(* IEC 61131-3 sources: Trae_CLoudTest/_archive/2026-04-25_全局规范修订V4.1.0/旧版程序文件 (part 2) *)

(* ---- FB_打胶机送料机构_V4.0.0.st ---- *)
//==============================================================================
// 边框缓存机 PLC程序 - 打胶机送料机构纯逻辑功能块
// 版本: V4.0.0
// 项目: DJ-2026-005 边框缓存机
// 编制日期: 2026-04-23
// 遵循规范: IEC 61131-3, 810_PLC编程规范_DEV-V1.0.0
// 说明: 纯逻辑功能块 - 打胶机送料机构独立控制(不包含任何X/Y/M/D地址引用)
//       所有输入来自主控(已映射的逻辑变量), 所有输出给主控(由主控映射到Y地址)
//
// 核心工艺:
//   接收取放料机构的放料完成信号后, X2轴移动到打胶机取料位置
//   等待打胶机允许送料 -> 发送允许抓料信号 -> 等待打胶机取料完成
//   返回待机位置, 循环执行
//
// 架构特点:
//   - 纯逻辑块: 不包含任何X/Y/M/D地址引用
//   - 数据解耦: 通过逻辑变量接口与主控交互
//   - 6步状态机: 完整的自动送料循环控制
//   - 故障安全: 内置超时保护、伺服故障检测、安全区冲突检测
//   - 安全区管理: 与取放料机构的区域互锁, 防止机械碰撞
//   - 完全自包含, 无外部物理地址依赖
//==============================================================================

//==============================================================================
// 功能块: FB_1004_GlueMachineFeeder_BufferFraming - 打胶机送料机构纯逻辑控制
// 功能:
//   1. 自动模式状态机(6步完整送料循环)
//   2. 手动模式控制(X2轴点动前/后)
//   3. 初始化流程(伺服使能、状态清零)
//   4. 块内报警检测与处理(5种报警类型, 201~299段)
//   5. 安全区逻辑(与取放料机构的区域互锁)
//   6. 完全自包含, 无外部物理地址依赖
//==============================================================================
FUNCTION_BLOCK FB_1004_GlueMachineFeeder_BufferFraming

VAR_INPUT
    (*==========================================================================
      一、系统控制信号 (来自主控/HMI M区)
      ==========================================================================*)
    i_b使能               : BOOL;    // 总使能信号(主控系统就绪后置位)

    (*-------------------------------------------------------------------------
      模式选择 (互斥信号,来自HMI M区)
      -------------------------------------------------------------------------*)
    i_b自动模式           : BOOL;    // 自动运行模式选择
    i_b手动模式           : BOOL;    // 手动调试模式选择

    (*-------------------------------------------------------------------------
      操作按钮 (来自HMI,边沿触发或电平有效)
      -------------------------------------------------------------------------*)
    i_b启动               : BOOL;    // 自动循环启动按钮(上升沿触发)
    i_b停止               : BOOL;    // 自动循环停止按钮(电平有效)
    i_b复位               : BOOL;    // 故障复位/初始化按钮(电平有效)

    (*==========================================================================
      二、手动操作信号 (2个BOOL,来自HMI)
      注: 本功能块仅控制X2轴(打胶机送料方向的水平轴)
      ==========================================================================*)
    (*--- X2轴伺服点动控制 (2个) ---*)
    i_bX2轴点动前         : BOOL;    // 手动-X2轴向前点动(去打胶机取料位置方向)
    i_bX2轴点动后         : BOOL;    // 手动-X2轴向后点动(返回待机位置方向)

    (*==========================================================================
      三、工艺参数 (来自HMI设定或配方, REAL类型)
      ==========================================================================*)
    i_r送料速度           : REAL;    // X2轴送料运动速度(mm/s或%)
    i_r待机位置           : REAL;    // X2轴待机位置坐标(mm, 安全等待位置)
    i_r取料位置           : REAL;    // X2轴取料位置坐标(mm, 打胶机取料口位置)

    (*==========================================================================
      四、传感器输入 (4个BOOL,全部来自主控IO映射)
      注: 本功能块不直接读取X地址, 所有传感器由主控映射后传入
      仅涉及X2轴相关传感器
      ==========================================================================*)
    (*--- X2轴伺服状态信号 ---*)
    i_bX2轴_原点           : BOOL;    // X2轴伺服原点信号(Home/ORG)
    i_bX2轴_正向限位       : BOOL;    // X2轴正向限位(去打胶机侧限位)
    i_bX2轴_反向限位       : BOOL;    // X2轴反向限位(待机位侧限位)
    i_bX2轴_伺服故障       : BOOL;    // X2轴伺服驱动器故障(ALM输出)

    (*==========================================================================
      五、打胶机交互信号 (2个BOOL,已由主控做IO映射)
      注: 这些是来自外部打胶机的硬接线信号, 由主控完成IO映射
      ==========================================================================*)
    i_b打胶机允许送料     : BOOL;    // 打胶机允许送料信号(对应物理地址X76)
                                    // TRUE=打胶机准备好可以接收边框
    i_b打胶机取料完成     : BOOL;    // 打胶机取料完成信号(对应物理地址X102)
                                    // TRUE=打胶机已完成边框抓取

    (*==========================================================================
      六、上游信号 (1个BOOL,来自取放料机构)
      ==========================================================================*)
    i_b取放料_放料完成    : BOOL;    // 取放料机构放料完成信号
                                    // TRUE=取放料机构已完成放料并移出安全区
END_VAR

VAR_OUTPUT
    (*==========================================================================
      一、执行器请求输出 (给主控, 由主控映射到Y地址)
      ==========================================================================*)

    (*--- 给打胶机的输出信号 ---*)
    o_b允许抓料            : BOOL;    // 允许抓料信号 -> 主控映射到Y44
                                    // 通知打胶机可以抓取边框(本站已到位且准备好)

    (*--- X2轴运动请求输出 (给主控驱动脉冲输出) ---*)
    o_bX2轴请求前移       : BOOL;    // X2轴向前移动请求(去打胶机取料位置)
    o_bX2轴请求后移       : BOOL;    // X2轴向后移动请求(返回待机位置)

    (*--- 安全区管理信号 ---*)
    o_b安全区信号          : BOOL;    // 安全区信号 -> 主控映射到Y47
                                    // TRUE=取放料机构在安全区外(打胶机可进入)
                                    // FALSE=取放料机构在工作区(禁止打胶机进入)

    (*==========================================================================
      二、状态/HMI显示输出
      ==========================================================================*)
    o_b运行中             : BOOL;    // 本站正在自动运行
    o_b故障               : BOOL;    // 本站有故障(任一报警激活)
    o_i当前状态           : INT;     // 当前状态机步序(0~5, 99=故障)
    o_rX2轴当前位置       : REAL;    // X2轴当前位置反馈(mm, 来自主控映射)

    (*==========================================================================
      三、报警输出 (给公共报警管理器)
      ==========================================================================*)
    o_i本站报警代码       : INT;     // 本站当前有效报警代码(0=无报警, 201~299=报警类型)
END_VAR

(*==============================================================================
 内部变量定义
 ==============================================================================*)
VAR
    (*--------------------------------------------------------------------------
      一、状态机核心变量
      --------------------------------------------------------------------------*)
    s_i步序               : INT;     // 当前状态机步序(0~5)
    s_b运行中             : BOOL;    // 自动运行中标志
    s_b故障               : BOOL;    // 故障标志
    s_b启动触发           : BOOL;    // 启动信号锁存(防重复触发)

    (*--- X2轴运动请求标志 (给主控处理脉冲输出) ---*)
    s_bX2轴请求前移       : BOOL;    // X2轴向前移动请求(去取料位置)
    s_bX2轴请求后移       : BOOL;    // X2轴向后移动请求(返回待机位置)
    s_bX2轴在待机位       : BOOL;    // X2轴是否在待机位置标志(由主控反馈)
    s_bX2轴在取料位       : BOOL;    // X2轴是否在取料位置标志(由主控反馈)

    (*--- 安全区管理变量 ---*)
    s_b取放料曾工作      : BOOL;    // 取放料机构曾经工作过标志(用于安全区判断)
    s_b上次放料完成      : BOOL;    // 上次扫描周期的放料完成状态(用于上升沿检测)

    (*--- 打胶机通讯超时检测 ---*)
    s_t通讯超时定时器     : TON;     // 打胶机响应超时检测定时器
    s_b等待打胶机响应     : BOOL;    // 正在等待打胶机响应标志

    (*--------------------------------------------------------------------------
      二、定时器 (覆盖所有时序需求)
      --------------------------------------------------------------------------*)
    s_t动作定时器         : TON;     // 通用动作等待定时器(X2轴移动等)
    s_t初始化定时器       : TON;     // 初始化总超时定时器
    s_t抓料保持定时器     : TON;     // 允许抓料信号保持定时器

    (*--------------------------------------------------------------------------
      三、系统级内部变量
      --------------------------------------------------------------------------*)
    s_b初始化完成         : BOOL;    // 上电初始化完成标志
    s_b初始化中           : BOOL;    // 正在执行初始化

    (*--- 报警相关 ---*)
    s_i活跃报警           : INT;     // 当前最高优先级报警代码

    (*--- 手动操作互锁 ---*)
    s_b手动允许           : BOOL;    // 允许手动操作标志
END_VAR

(*==============================================================================
 常量定义 (状态机步序 + 报警码 + 定时参数)
 ==============================================================================*)
VAR CONSTANT
    (*--------------------------------------------------------------------------
      状态机步序常量 (6步: 0空闲 + 5工作步)
      核心工艺: 接收放料完成 -> 移动到取料位 -> 等待允许 -> 抓料 -> 返回待机
      --------------------------------------------------------------------------*)
    STP_空闲              : INT := 0;   // 空闲/待机位置
    STP_等待放料完成      : INT := 1;   // 等待取放料机构放料完成
    STP_移动到取料位置    : INT := 2;   // X2轴移动到打胶机取料位置
    STP_等待允许送料      : INT := 3;   // 等待打胶机允许送料信号
    STP_发送允许抓料      : INT := 4;   // 发送允许抓料+等待打胶机取料完成
    STP_返回待机位置      : INT := 5;   // X2轴返回待机位置

    (*--------------------------------------------------------------------------
      报警码常量 (201~299段, 0=无报警)
      与取放料机构(101~199段)、其他设备错开, 便于公共报警管理器区分来源
      --------------------------------------------------------------------------*)
    ALM_通讯超时          : INT := 201;  // 通讯超时(打胶机无响应)
    ALM_安全区冲突        : INT := 202;  // 安全区冲突(取放料未离开)
    ALM_X2轴伺服故障      : INT := 203;  // X2轴伺服驱动器故障
    ALM_X2轴移动超时      : INT := 204;  // X2轴移动超时(未到达目标位置)
    ALM_取料位置到达超时  : INT := 205;  // 取料位置到达超时(步骤2专用)

    (*--------------------------------------------------------------------------
      默认定时参数 (单位: ms 或 s, 可通过输入参数覆盖)
      --------------------------------------------------------------------------*)
    T_DEF_移动超时时间    : INT := 5000;    // X2轴移动超时保护(5s)
    T_DEF_通讯超时时间    : INT := 10000;   // 打胶机响应超时(10s)
    T_DEF_抓料保持时间    : INT := 500;     // 允许抓料信号保持时间(500ms)
    T_DEF_初始化超时      : INT := 10000;   // 初始化总超时(10s)
END_VAR

(*==============================================================================
 主程序开始
 ==============================================================================*)

//==============================================================================
// 第一部分: 使能与初始化处理
//==============================================================================

(*--- 使能失效时的安全处理: 全部输出归零, 状态复位 ---*)
IF NOT i_b使能 THEN
    (
    (* 清零所有执行器输出 *)
    o_b允许抓料            := FALSE;
    o_b安全区信号          := FALSE;
    o_bX2轴请求前移       := FALSE;
    o_bX2轴请求后移       := FALSE;

    (* 清零所有状态 *)
    s_i步序               := STP_空闲
    s_b运行中             := FALSE;
    s_b故障               := FALSE;
    s_b启动触发           := FALSE;

    (* 清零运动请求 *)
    s_bX2轴请求前移       := FALSE;
    s_bX2轴请求后移       := FALSE;
    s_bX2轴在待机位       := FALSE;
    s_bX2轴在取料位       := FALSE;

    (* 清零安全区变量 *)
    s_b取放料曾工作      := FALSE;
    s_b上次放料完成      := FALSE;
    s_b等待打胶机响应     := FALSE;

    (* 清零报警 *)
    s_i活跃报警           := 0;
    o_i本站报警代码       := 0;
    o_b故障               := FALSE;
    s_b初始化完成         := FALSE;
    s_b初始化中           := FALSE;

    (* 清零状态输出 *)
    o_b运行中             := FALSE;
    o_i当前状态           := STP_空闲;

    (* 停止所有定时器 *)
    s_t动作定时器(IN := FALSE);
    s_t通讯超时定时器(IN := FALSE);
    s_t初始化定时器(IN := FALSE);
    s_t抓料保持定时器(IN := FALSE);

    RETURN;  (* 退出功能块, 不执行后续逻辑 *)
END_IF;

//==============================================================================
// 第二部分: 初始化流程 (上电或复位后首次使能时执行)
//==============================================================================

IF NOT s_b初始化完成 THEN
    s_b初始化中 := TRUE;

    (* 初始化定时器: 防止初始化卡死 *)
    s_t初始化定时器(IN := TRUE, PT := T_DEF_初始化超时);

    (* 初始化动作:
       1. 所有输出回到安全状态(禁止抓料, 安全区FALSE)
       2. 伺服使能准备(实际使能由主控统一协调)
       3. 状态清零
    *)

    (* 安全输出状态: 禁止抓料, 安全区默认FALSE(保守策略) *)
    o_b允许抓料            := FALSE;
    o_b安全区信号          := FALSE;
    o_bX2轴请求前移       := FALSE;
    o_bX2轴请求后移       := FALSE;

    (* 步序归零 *)
    s_i步序               := STP_空闲;
    s_b故障               := FALSE;
    s_i活跃报警           := 0;

    (* 检查初始化条件:
       X2轴伺服无故障 AND (已在原点 OR 超时强制完成)
       允许在有非关键报警情况下继续, 报警单独处理
    *)
    IF (NOT i_bX2轴_伺服故障) OR s_t初始化定时器.Q THEN
        (* 初始化完成 或 超时强制完成(伺服故障会单独报203号报警) *)
        s_b初始化完成 := TRUE;
        s_b初始化中 := FALSE;
        s_t初始化定时器(IN := FALSE);

        (* 初始化完成后关闭输出(进入空闲态的安全状态) *)
        o_b允许抓料        := FALSE;
        o_b安全区信号      := FALSE;
        o_bX2轴请求前移   := FALSE;
        o_bX2轴请求后移   := FALSE;
    END_IF;

    (* 初始化期间不执行自动/手动逻辑 *)
    o_b运行中 := FALSE;
    o_i当前状态 := STP_空闲;
    RETURN;
END_IF;

//==============================================================================
// 第三部分: 安全区逻辑处理 (所有模式共用, 最高优先级之一)
//==============================================================================

(*--- 安全区核心逻辑 ---
   目的: 防止取放料机构和打胶机同时在工作区域造成碰撞
   原则: 取放料机构优先(它是主动方, 先放料后打胶机才能进来)

   判断依据:
   - i_b取放料_放料完成 = TRUE 表示取放料机构已完成放料并移出工作区
   - 当取放料机构正在工作时(放料完成=FALSE), 安全区应为FALSE
   - 只有当放料完成且确认离开后, 安全区才为TRUE
*)

(*--- 检测取放料机构工作状态的上升沿 ---*)
(* 当放料完成从FALSE变为TRUE时, 说明取放料机构刚完成工作并离开 *)
IF i_b取放料_放料完成 AND NOT s_b上次放料完成 THEN
    (* 放料完成的上升沿: 标记取放料机构曾工作过, 现在已离开 *)
    s_b取放料曾工作 := TRUE;
ELSIF NOT i_b取放料_放料完成 THEN
    (* 放料完成=FALSE: 取放料机构可能正在工作中或尚未开始 *)
    (* 如果之前有过放料完成又变为FALSE, 说明新的一轮开始了 *)
END_IF;

(*--- 更新上次状态(用于下次扫描周期的上升沿检测) ---*)
s_b上次放料完成 := i_b取放料_放料完成;

(*--- 安全区信号输出逻辑 ---*)
IF i_b取放料_放料完成 THEN
    (* 放料完成=TRUE: 取放料机构已离开工作区, 安全区开放 *)
    o_b安全区信号 := TRUE;
ELSE
    (* 放料完成=FALSE: 取放料机构可能还在工作区, 安全区关闭 *)
    o_b安全区信号 := FALSE;
END_IF;

//==============================================================================
// 第四部分: X2轴伺服故障检测 (所有模式共用, 最高优先级)
//==============================================================================

(*--- X2轴伺服故障检测 ---*)
IF i_bX2轴_伺服故障 THEN
    IF s_i活跃报警 <> ALM_X2轴伺服故障 THEN
        (* 新故障: 记录报警 *)
        s_i活跃报警 := ALM_X2轴伺服故障;
        s_b故障 := TRUE;
    END_IF;
    (* 伺服故障时立即停止X2轴运动请求 *)
    s_bX2轴请求前移   := FALSE;
    o_bX2轴请求前移   := FALSE;
    s_bX2轴请求后移   := FALSE;
    o_bX2轴请求后移   := FALSE;
ELSIF s_i活跃报警 = ALM_X2轴伺服故障 THEN
    (* 故障消失且当前只有此报警 -> 清除 *)
    s_i活跃报警 := 0;
    s_b故障 := FALSE;
END_IF;

//==============================================================================
// 第五部分: 模式分发 (自动/手动)
//==============================================================================

IF i_b自动模式 THEN
    (*==========================================================================
      自动模式: 执行6步送料状态机
      =========================================================================*)
    CALL_自动模式状态机();

ELSIF i_b手动模式 THEN
    (*==========================================================================
      手动模式: 执行手动点动控制(X2轴前后点动)
      =========================================================================*)
    CALL_手动模式控制();

ELSE
    (* 无效模式: 停止所有输出, 进入安全状态 *)
    o_b允许抓料            := FALSE;
    o_bX2轴请求前移       := FALSE;
    o_bX2轴请求后移       := FALSE;

    (* 如果不在故障态, 归零步序 *)
    IF NOT s_b故障 THEN
        s_i步序 := STP_空闲;
        s_b运行中 := FALSE;
    END_IF;
END_IF;

//==============================================================================
// 第六部分: 停止与复位处理
//==============================================================================

(*--- 全局停止: 停止自动循环, 保持当前位置 ---*)
IF i_b停止 THEN
    IF s_b运行中 AND NOT s_b故障 THEN
        (* 停止并复位到空闲 *)
        s_i步序 := STP_空闲;
        s_b运行中 := FALSE;
        s_b启动触发 := FALSE;

        (* 停止所有输出 *)
        o_b允许抓料            := FALSE;
        o_bX2轴请求前移       := FALSE;
        o_bX2轴请求后移       := FALSE;
        s_bX2轴请求前移       := FALSE;
        s_bX2轴请求后移       := FALSE;

        (* 停止定时器 *)
        s_t动作定时器(IN := FALSE);
        s_t通讯超时定时器(IN := FALSE);
        s_t抓料保持定时器(IN := FALSE);
        s_b等待打胶机响应     := FALSE;
    END_IF;
END_IF;

(*--- 全局复位: 清除所有报警和故障, 重新初始化 ---*)
IF i_b复位 THEN
    IF s_b故障 THEN
        (* 清除报警和故障标志 *)
        s_i活跃报警 := 0;
        s_b故障 := FALSE;
        o_i本站报警代码 := 0;

        (* 归零步序和计数器 *)
        s_i步序 := STP_空闲;
        s_b运行中 := FALSE;
        s_b启动触发 := FALSE;

        (* 安全输出状态: 全部归零 *)
        o_b允许抓料            := FALSE;
        o_bX2轴请求前移       := FALSE;
        o_bX2轴请求后移       := FALSE;
        s_bX2轴请求前移       := FALSE;
        s_bX2轴请求后移       := FALSE;
        s_bX2轴在待机位       := FALSE;
        s_bX2轴在取料位       := FALSE;

        (* 清零安全区变量 *)
        s_b取放料曾工作      := FALSE;
        s_b等待打胶机响应     := FALSE;

        (* 停止定时器 *)
        s_t动作定时器(IN := FALSE);
        s_t通讯超时定时器(IN := FALSE);
        s_t抓料保持定时器(IN := FALSE);

        (* 要求重新初始化 *)
        s_b初始化完成 := FALSE;
    END_IF;
END_IF;

//==============================================================================
// 第七部分: 状态输出汇总
//==============================================================================

(*--- 运行中标志 ---*)
o_b运行中 := s_b运行中;

(*--- 故障标志 ---*)
o_b故障 := s_b故障;

(*--- 当前状态码 ---*)
IF s_b故障 THEN
    o_i当前状态 := 99;  (* 故障状态显示99 *)
ELSE
    o_i当前状态 := s_i步序;
END_IF;

(*--- 本站报警代码 ---*)
o_i本站报警代码 := s_i活跃报警;

(*==============================================================================
 子程序: 自动模式状态机 (6步完整送料循环)
   核心工艺: 等待放料完成 -> X2轴移动到取料位 -> 等待允许 -> 抓料 -> 返回待机
   安全约束: 步骤1需要安全区信号为TRUE才能继续
  ==============================================================================*)
METHOD CALL_自动模式状态机 : VOID

    (*--- 故障时不执行状态机 ---*)
    IF s_b故障 THEN
        s_b运行中 := FALSE;
        (* 故障安全输出: 全部停止 *)
        o_b允许抓料            := FALSE;
        o_bX2轴请求前移       := FALSE;
        o_bX2轴请求后移       := FALSE;
        s_bX2轴请求前移       := FALSE;
        s_bX2轴请求后移       := FALSE;
        s_t动作定时器(IN := FALSE);
        s_t通讯超时定时器(IN := FALSE);
        s_t抓料保持定时器(IN := FALSE);
        s_b等待打胶机响应     := FALSE;
        RETURN;
    END_IF;

    (*--- 启动触发检测 (上升沿) ---*)
    IF i_b启动 AND NOT s_b启动触发 THEN
        s_b启动触发 := TRUE;
    END_IF;

    (*--- 单例状态机 (全局唯一, 因为只有一个打胶机送料机构) ---*)
    CASE s_i步序 OF

    (*======================================================================
     步骤0: 空闲/待机位置
     等待启动触发, 收到启动后进入等待放料完成
     ======================================================================*)
    STP_空闲:
        s_b运行中 := FALSE;
        (* 安全输出状态: 全部归零 *)
        o_b允许抓料            := FALSE;
        o_bX2轴请求前移       := FALSE;
        o_bX2轴请求后移       := FALSE;
        s_bX2轴请求前移       := FALSE;
        s_bX2轴请求后移       := FALSE;
        s_b等待打胶机响应     := FALSE;

        (* 启动条件: 收到启动触发 *)
        IF s_b启动触发 THEN
            s_i步序 := STP_等待放料完成;
            s_b运行中 := TRUE;
        END_IF;

    (*======================================================================
     步骤1: 等待取放料放料完成
     等待取放料机构的放料完成信号(即安全区开放)
     条件: i_b取放料_放料完成 = TRUE
     ======================================================================*)
    STP_等待放料完成:
        (* 保持安全输出状态 *)
        o_b允许抓料            := FALSE;
        o_bX2轴请求前移       := FALSE;
        o_bX2轴请求后移       := FALSE;
        s_bX2轴请求前移       := FALSE;
        s_bX2轴请求后移       := FALSE;

        (* 等待条件: 取放料机构放料完成(安全区开放) *)
        IF i_b取放料_放料完成 THEN
            (* 放料完成, 可以开始移动到取料位置 *)
            s_i步序 := STP_移动到取料位置;
            (* 启动移动超时定时器 *)
            s_t动作定时器(IN := TRUE, PT := T_DEF_移动超时时间);
            (* 请求X2轴向前移动(去打胶机取料位置) *)
            s_bX2轴请求前移   := TRUE;
            o_bX2轴请求前移   := TRUE;
            s_bX2轴请求后移   := FALSE;
            o_bX2轴请求后移   := FALSE;
            s_bX2轴在待机位   := FALSE;
        END_IF;

        (* 注意: 此步骤没有独立的超时报警, 因为等待上游信号是正常行为
           超时保护由公共层或操作员手动停止处理 *)

    (*======================================================================
     步骤2: 移动到打胶机取料位置 (X2轴水平移动)
     X2轴向前移动到打胶机取料口位置
     等待X2轴到达取料位置或超时
     注: X2轴的实际脉冲输出由主控根据请求标志处理
     ======================================================================*)
    STP_移动到取料位置:
        (* 保持X2轴前移请求 *)
        s_bX2轴请求前移   := TRUE;
        o_bX2轴请求前移   := TRUE;
        s_bX2轴请求后移   := FALSE;
        o_bX2轴请求后移   := FALSE;

        (* 到达取料位置的判断:
           由主控在X2轴到达目标位置后置位s_bX2轴在取料位
           或通过位置判断(i_rX2轴当前位置接近i_r取料位置)
        *)
        IF s_bX2轴在取料位 THEN
            (* 到达取料位置, 转入等待打胶机允许送料 *)
            s_t动作定时器(IN := FALSE);
            s_bX2轴请求前移   := FALSE;
            o_bX2轴请求前移   := FALSE;
            s_bX2轴在取料位   := TRUE;
            s_i步序 := STP_等待允许送料;
            (* 启动通讯超时定时器(等待打胶机响应) *)
            s_t通讯超时定时器(IN := TRUE, PT := T_DEF_通讯超时时间);
            s_b等待打胶机响应 := TRUE;
        ELSIF s_t动作定时器.Q THEN
            (* 超时: X2轴未在规定时间内到达取料位置 *)
            s_t动作定时器(IN := FALSE);
            s_i活跃报警 := ALM_X2轴移动超时;
            s_b故障 := TRUE;
            s_bX2轴请求前移   := FALSE;
            o_bX2轴请求前移   := FALSE;
            s_i步序 := STP_空闲;
            s_b运行中 := FALSE;
            s_b启动触发 := FALSE;
            s_b等待打胶机响应 := FALSE;
        END_IF;

    (*======================================================================
     步骤3: 等待打胶机允许送料
     等待打胶机发出允许送料信号(i_b打胶机允许送料=TRUE)
     同时监控通讯超时
     ======================================================================*)
    STP_等待允许送料:
        (* 保持当前状态, 等待打胶机响应 *)
        s_bX2轴请求前移   := FALSE;
        o_bX2轴请求前移   := FALSE;
        s_bX2轴请求后移   := FALSE;
        o_bX2轴请求后移   := FALSE;
        o_b允许抓料        := FALSE;

        (* 检查打胶机允许送料信号 *)
        IF i_b打胶机允许送料 THEN
            (* 打胶机允许送料, 转入发送允许抓料步骤 *)
            s_t通讯超时定时器(IN := FALSE);
            s_b等待打胶机响应 := FALSE;
            s_i步序 := STP_发送允许抓料;
            (* 启动抓料保持定时器和通讯超时定时器(等待取料完成) *)
            s_t抓料保持定时器(IN := TRUE, PT := T_DEF_抓料保持时间);
            s_t通讯超时定时器(IN := TRUE, PT := T_DEF_通讯超时时间);
            s_b等待打胶机响应 := TRUE;
            (* 发送允许抓料信号 *)
            o_b允许抓料 := TRUE;
        ELSIF s_t通讯超时定时器.Q THEN
            (* 超时: 打胶机长时间无响应 *)
            s_t通讯超时定时器(IN := FALSE);
            s_i活跃报警 := ALM_通讯超时;
            s_b故障 := TRUE;
            o_b允许抓料 := FALSE;
            s_b等待打胶机响应 := FALSE;
            s_i步序 := STP_空闲;
            s_b运行中 := FALSE;
            s_b启动触发 := FALSE;
        END_IF;

    (*======================================================================
     步骤4: 发送允许抓料 + 等待打胶机取料完成
     保持允许抓料信号, 等待打胶机完成取料动作
     ======================================================================*)
    STP_发送允许抓料:
        (* 保持允许抓料输出 *)
        o_b允许抓料 := TRUE;
        s_bX2轴请求前移 := FALSE;
        o_bX2轴请求前移 := FALSE;
        s_bX2轴请求后移 := FALSE;
        o_bX2轴请求后移 := FALSE;

        (* 检查打胶机取料完成信号 *)
        IF i_b打胶机取料完成 THEN
            (* 打胶机取料完成, 转入返回待机位置 *)
            s_t通讯超时定时器(IN := FALSE);
            s_t抓料保持定时器(IN := FALSE);
            s_b等待打胶机响应 := FALSE;
            (* 保持一段时间的允许抓料信号后关闭 *)
            (* 或者立即关闭, 根据实际工艺需求 *)
            o_b允许抓料 := FALSE;
            s_i步序 := STP_返回待机位置;
            (* 启动返回移动定时器 *)
            s_t动作定时器(IN := TRUE, PT := T_DEF_移动超时时间);
            (* 请求X2轴向后移动(返回待机位置) *)
            s_bX2轴请求前移   := FALSE;
            o_bX2轴请求前移   := FALSE;
            s_bX2轴请求后移   := TRUE;
            o_bX2轴请求后移   := TRUE;
            s_bX2轴在取料位   := FALSE;
        ELSIF s_t通讯超时定时器.Q THEN
            (* 超时: 打胶机取料超时 *)
            s_t通讯超时定时器(IN := FALSE);
            s_t抓料保持定时器(IN := FALSE);
            s_i活跃报警 := ALM_通讯超时;
            s_b故障 := TRUE;
            o_b允许抓料 := FALSE;
            s_b等待打胶机响应 := FALSE;
            s_bX2轴请求后移 := FALSE;
            o_bX2轴请求后移 := FALSE;
            s_i步序 := STP_空闲;
            s_b运行中 := FALSE;
            s_b启动触发 := FALSE;
        END_IF;

    (*======================================================================
     步骤5: 返回待机位置 (X2轴水平移动回待机位)
     X2轴向后移动回到待机位置(安全等待位置)
     等待X2轴到达待机位置或超时
     完成后回到步骤1, 继续下一轮循环
     ======================================================================*)
    STP_返回待机位置:
        (* 保持X2轴后移请求 *)
        s_bX2轴请求前移   := FALSE;
        o_bX2轴请求前移   := FALSE;
        s_bX2轴请求后移   := TRUE;
        o_bX2轴请求后移   := TRUE;

        (* 到达待机位置的判断:
           由主控在X2轴到达目标位置后置位s_bX2轴在待机位
           或通过位置判断(i_rX2轴当前位置接近i_r待机位置)
        *)
        IF s_bX2轴在待机位 THEN
            (* 到达待机位置, 完成一轮循环, 回到等待放料完成 *)
            s_t动作定时器(IN := FALSE);
            s_bX2轴请求后移   := FALSE;
            o_bX2轴请求后移   := FALSE;
            s_bX2轴在待机位   := TRUE;
            s_i步序 := STP_等待放料完成;  (* 回到步骤1, 继续循环 *)
            (* 不重置s_b启动触发, 保持连续循环 *)
        ELSIF s_t动作定时器.Q THEN
            (* 超时: X2轴未在规定时间内返回待机位置 *)
            s_t动作定时器(IN := FALSE);
            s_i活跃报警 := ALM_X2轴移动超时;
            s_b故障 := TRUE;
            s_bX2轴请求后移   := FALSE;
            o_bX2轴请求后移   := FALSE;
            s_i步序 := STP_空闲;
            s_b运行中 := FALSE;
            s_b启动触发 := FALSE;
        END_IF;

    ELSE
        (* 无效步序: 强制归零 *)
        s_i步序 := STP_空闲;
        s_b运行中 := FALSE;

    END_CASE;

(*==============================================================================
 子程序: 手动模式控制 (X2轴点动前/后, 带互锁和安全限制)
  ==============================================================================*)
METHOD CALL_手动模式控制 : VOID

    (*--- 故障时禁止手动操作 ---*)
    IF s_b故障 THEN
        s_b手动允许 := FALSE;
        o_b允许抓料            := FALSE;
        s_bX2轴请求前移       := FALSE;
        s_bX2轴请求后移       := FALSE;
        s_i步序 := STP_空闲;
        s_b运行中 := FALSE;
        RETURN;
    END_IF;

    s_b手动允许 := TRUE;
    s_b运行中 := FALSE;
    s_i步序 := STP_空闲;  (* 手动模式下步序显示为空闲 *)
    o_b允许抓料 := FALSE;   (* 手动模式下不允许自动抓料 *)

    (*======================================================================
     手动操作 - X2轴伺服点动控制 (前/后互锁)
     注意: 伺服的点动脉冲输出由主控根据请求标志处理
     本功能块只输出请求标志
     ======================================================================*)

    (*--- X2轴点动: 前/后互锁 ---*)
    IF i_bX2轴点动前 AND NOT i_bX2轴点动后 THEN
        (* X2轴向前点动(去打胶机取料位置方向) *)
        (* 检查是否已到正向限位 *)
        IF NOT i_bX2轴_正向限位 THEN
            s_bX2轴请求前移 := TRUE;
            o_bX2轴请求前移 := TRUE;
            s_bX2轴请求后移 := FALSE;
            o_bX2轴请求后移 := FALSE;
        END_IF;
    ELSIF i_bX2轴点动后 AND NOT i_bX2轴点动前 THEN
        (* X2轴向后点动(返回待机位置方向) *)
        (* 检查是否已到反向限位 *)
        IF NOT i_bX2轴_反向限位 THEN
            s_bX2轴请求后移 := TRUE;
            o_bX2轴请求后移 := TRUE;
            s_bX2轴请求前移 := FALSE;
            o_bX2轴请求前移 := FALSE;
        END_IF;
    ELSE
        (* 无X2轴点动操作 *)
        s_bX2轴请求前移 := FALSE;
        o_bX2轴请求前移 := FALSE;
        s_bX2轴请求后移 := FALSE;
        o_bX2轴请求后移 := FALSE;
    END_IF;

END_FUNCTION_BLOCK

//==============================================================================
// 程序结束
//==============================================================================

(* ---- 主控程序_V4.0.0.st ---- *)
//==============================================================================
// 边框缓存机 PLC程序 - 主控程序 (V4.0.0架构)
// 版本: V4.0.0
// 项目: DJ-2026-005 边框缓存机
// 编制日期: 2026-04-23
// 更新日期: 2026-04-24 (新增打胶机/组框机交互接口预留)
// 遵循规范: IEC 61131-3, 810_PLC编程规范_DEV-V1.0.0
//
// 说明:
//   主控程序是系统的核心协调组件,承担以下职责:
//   1. IO映射: X地址->逻辑变量(传感器输入), 逻辑变量->Y地址(执行器输出)
//   2. HMI数据交互: M/D区读取(操作指令/参数设定), M/D区回写(状态/报警)
//   3. 外部设备交互:
//      - 下游打胶机: 允许送料(X76), 取料完成(X102), 故障/急停联锁
//      - 上游组框机: 允许送料, 有料请求, 开门互锁, 安全联锁 (预留接口)
//   4. 工站实例化与连接: 实例化4个功能块并按工艺顺序调用
//   5. 报警汇总: 调用公共报警管理器,汇总三工站报警并写入D区
//
// 架构特点:
//   - 纯协调层: 不包含任何业务逻辑(状态机/自动手动判断在工站内部)
//   - 数据桥梁: 连接物理IO层(X/Y)与逻辑层(功能块接口变量)
//   - 设备协调: 处理上下游设备的握手、联锁、互锁信号
//   - 执行顺序严格: 输入映射->外部信号处理->工站调用->输出映射
//   - 接口预留: 组框机信号使用占位符, 待现场确定物理地址后激活
//
// 外部设备交互协议:
//   ┌───────────┐    边框流入     ┌──────────────┐    边框流出    ┌───────────┐
//   │           │ ──────────────> │              │ ──────────────> │           │
//   │  组框机   │               │  边框缓存机   │               │  打胶机   │
//   │ (上游)    │ <────────────── │   (本设备)    │ <────────────── │ (下游)    │
//   │           │   控制/状态信号 │              │   控制/状态信号 │           │
//   └───────────┘               └──────────────┘               └───────────┘
//
// 执行顺序(每个扫描周期):
//   Step1: IO映射输入 (X地址 -> 逻辑变量, 含打胶机/组框机DI)
//   Step2: HMI数据读取 (M/D区 -> 逻辑变量)
//   Step3: 外部设备信号处理 (打胶机有效性检查 + 组框机安全联锁)
//   Step4: 调用fb四层输送机 (传入所有输入, 接收所有输出)
//   Step5: 调用fb取放料机构 (传入含上游信号的输入)
//   Step6: 调用fb打胶机送料机构 (传入含上游+打胶机信号的输入)
//   Step7: 调用fb公共报警 (汇总各工站报警)
//   Step8: IO映射输出 (逻辑变量 -> Y地址, 含打胶机/组框机DO)
//   Step9: HMI状态回写 (逻辑变量 -> M/D区)
//   Step10: 报警D区回写 (公共报警输出 -> D400起始)
//==============================================================================

PROGRAM 主控程序

VAR
    // ==========================================================================
    // 一、工站实例声明 (4个纯逻辑功能块, 无物理地址依赖)
    // ==========================================================================

    (*--- 工站1: 四层输送机 (独立控制4层分料/输送) ---*)
    fb四层输送机      : FB_1001_Conveyor4Layer_BufferFraming;

    (*--- 工站2: 取放料机构 (Z轴升降+X1轴横移+夹爪控制) ---*)
    fb取放料机构      : FB_1003_PickPlace_BufferFraming;

    (*--- 工站3: 打胶机送料机构 (X2轴横移+打胶机交互) ---*)
    fb打胶机送料机构   : FB_1004_GlueMachineFeeder_BufferFraming;

    (*--- 工站4: 公共报警管理器 (汇总三工站报警+MES队列) ---*)
    fb公共报警        : FB_2001_CommonAlarm_AllStation;

    // ==========================================================================
    // 二、四层输送机 - 传感器输入映射 (X地址 -> 逻辑变量)
    // 注: 物理地址来自DI扩展模块3(DI3)和DI扩展模块4(DI4)
    //     DI3: X0-X17对应4层(L4)和3层(L3), DI4: X0-X17对应2层(L2)和1层(L1)
    //     数组索引: [1]=第1层(底层/L1), [4]=第4层(顶层/L4)
    // ==========================================================================

    (*--- 分料前感应器: 检测材料是否到达分料工位入口 ---*)
    (* DI4:X11=L1, DI4:X1=L2, DI3:X11=L3, DI3:X0=L4 *)
    i_bLx_分料前感应器    : ARRAY[1..4] OF BOOL;   // X51,X61,X71,X81

    (*--- 到位感应器1/2: 双传感器冗余检测材料到位 ---*)
    (* DI4:X12/X13=L1, DI4:X2/X3=L2, DI3:X12/X13=L3, DI3:X2/X3=L4 *)
    i_bLx_到位感应器1     : ARRAY[1..4] OF BOOL;   // X52,X62,X72,X82
    i_bLx_到位感应器2     : ARRAY[1..4] OF BOOL;   // X53,X63,X73,X83

    (*--- 阻挡气缸位置反馈 ---*)
    (* DI4:X14/X15=L1, DI4:X4/X5=L2, DI3:X14/X15=L3, DI3:X4/X5=L4 *)
    i_bLx_阻挡气缸上位    : ARRAY[1..4] OF BOOL;   // X54,X64,X74,X84
    i_bLx_阻挡气缸下位    : ARRAY[1..4] OF BOOL;   // X55,X65,X75,X85

    (*--- 分料气缸位置反馈 ---*)
    (* DI4:X16/X17=L1, DI4:X6/X7=L2, DI3:X16/X17=L3, DI3:X6/X7=L4 *)
    i_bLx_分料气缸上位    : ARRAY[1..4] OF BOOL;   // X56,X66,X76,X86
    i_bLx_分料气缸下位    : ARRAY[1..4] OF BOOL;   // X57,X67,X77,X87

    // ==========================================================================
    // 三、四层输送机 - 执行器输出映射 (逻辑变量 -> Y地址)
    // 注: 物理地址来自DO扩展模块1(DO1)和DO扩展模块2(DO2)
    //     DO1: Y0-Y5=L4, Y10-Y15=L3 | DO2: Y0-Y5=L2, Y10-Y15=L1
    // ==========================================================================

    (*--- 阻挡电磁阀: TRUE=下降(阻挡), FALSE=上升(释放) ---*)
    (* DO2:Y10=L1, DO2:Y0=L2, DO1:Y10=L3, DO1:Y0=L4 *)
    q_bLx_阻挡电磁阀      : ARRAY[1..4] OF BOOL;   // Y20,Y21,Y22,Y23

    (*--- 分料电磁阀: TRUE=推出(分料), FALSE=复位 ---*)
    (* DO2:Y11=L1, DO2:Y1=L2, DO1:Y11=L3, DO1:Y1=L4 *)
    q_bLx_分料电磁阀      : ARRAY[1..4] OF BOOL;   // Y24,Y25,Y26,Y27

    (*--- 输送带正转 ---*)
    (* DO2:Y12=L1, DO2:Y2=L2, DO1:Y12=L3, DO1:Y2=L4 *)
    q_bLx_输送带正转      : ARRAY[1..4] OF BOOL;   // Y28,Y29,Y30,Y31

    (*--- 输送带慢速 (精确定位用) ---*)
    (* DO2:Y13=L1, DO2:Y3=L2, DO1:Y13=L3, DO1:Y3=L4 *)
    q_bLx_输送带慢速      : ARRAY[1..4] OF BOOL;   // Y32,Y33,Y34,Y35

    (*--- 输送带反转 (预留) ---*)
    q_bLx_输送带反转     : ARRAY[1..4] OF BOOL;   // 预留: Y24,Y30,Y36,Y42

    // ==========================================================================
    // 四、取放料机构 - 传感器输入映射
    // 注: 物理地址来自远程IO_1(站号1, CC-Link Basic) + CPU本体(X0-X13)
    // ==========================================================================

    (*--- 气缸位置传感器 (10个磁性开关, 来自Remote_IO X0-X9) ---*)
    (* 升降气缸: 动点=下降到位, 原点=上升到位 *)
    i_b升降_动点          : BOOL;   // Remote_X0
    i_b升降_原点          : BOOL;   // Remote_X1

    (* 前夹紧气缸: 动点=夹紧到位, 原点=松开到位 *)
    i_b前夹紧_动点        : BOOL;   // Remote_X2
    i_b前夹紧_原点        : BOOL;   // Remote_X3

    (* 后夹紧气缸: 动点=夹紧到位, 原点=松开到位 *)
    i_b后夹紧_动点        : BOOL;   // Remote_X4
    i_b后夹紧_原点        : BOOL;   // Remote_X5

    (* 前夹紧2气缸: 第二组前夹爪 *)
    i_b前夹紧2_动点       : BOOL;   // Remote_X6
    i_b前夹紧2_原点       : BOOL;   // Remote_X7

    (* 后夹紧2气缸: 第二组后夹爪 *)
    i_b后夹紧2_动点       : BOOL;   // Remote_X8
    i_b后夹紧2_原点       : BOOL;   // Remote_X9

    (*--- 产品检测传感器 (4个光电传感器, 来自Remote_IO XC-XF) ---*)
    (* 一次取两根边框: 长边×2 + 短边×2 *)
    i_b长边1检测          : BOOL;   // Remote_XC
    i_b长边2检测          : BOOL;   // Remote_XD
    i_b短边1检测          : BOOL;   // Remote_XE
    i_b短边2检测          : BOOL;   // Remote_XF

    (*--- 伺服轴状态信号 (12个, 来自CPU本体X0-X13) ---*)
    (* 原点信号 *)
    i_bZ轴_原点           : BOOL;   // X0
    i_bX1轴_原点          : BOOL;   // X1
    i_bX2轴_原点          : BOOL;   // X2

    (* 伺服故障报警 *)
    i_bZ轴_伺服故障       : BOOL;   // X11
    i_bX1轴_伺服故障      : BOOL;   // X12
    i_bX2轴_伺服故障      : BOOL;   // X13

    (* 限位开关信号 *)
    i_bZ轴_正向限位       : BOOL;   // X3
    i_bZ轴_反向限位       : BOOL;   // X4
    i_bX1轴_正向限位      : BOOL;   // X5
    i_bX1轴_反向限位      : BOOL;   // X6
    i_bX2轴_正向限位      : BOOL;   // X7
    i_bX2轴_反向限位      : BOOL;   // X10

    // ==========================================================================
    // 五、取放料机构 - 执行器输出映射
    // ==========================================================================

    (*--- 气缸控制输出 (6个BOOL, 映射到Remote_IO Y10-Y15) ---*)
    (* 升降气缸: 上升/下降双电磁阀 *)
    q_b升降_上升          : BOOL;   // -> Remote_Y10
    q_b升降_下降          : BOOL;   // -> Remote_Y11

    (* 前夹紧气缸: 夹紧/松开双电磁阀 *)
    q_b前夹紧_夹紧        : BOOL;   // -> Remote_Y12
    q_b前夹紧_松开        : BOOL;   // -> Remote_Y13

    (* 后夹紧气缸: 夹紧/松开双电磁阀 *)
    q_b后夹紧_夹紧        : BOOL;   // -> Remote_Y14
    q_b后夹紧_松开        : BOOL;   // -> Remote_Y15

    (*--- 伺服控制输出 (3个BOOL, 仅Z轴由本程序直接映射到CPU Y地址) ---*)
    (* 注: X1轴/X2轴的脉冲输出由运动控制模块处理, 此处仅做标志传递 *)
    q_bZ轴_脉冲输出       : BOOL;   // -> Y0 (PULSE+)
    q_bZ轴_方向输出       : BOOL;   // -> Y1 (DIR+)
    q_bZ轴_伺服使能       : BOOL;   // -> Y2 (SERVO ON)

    // ==========================================================================
    // 六、打胶机信号映射 (下游设备: 接收边框并打胶)
    // ==========================================================================

    (*--- 打胶机输入信号 (来自CPU本体DI, 硬接线/通讯) ---*)
    i_b打胶机_自动中      : BOOL;   // %IX75  占位符: 打胶机自动运行中
    i_b打胶机_允许送料    : BOOL;   // %IX76  (已定义) 打胶机准备好可接收边框
    i_b打胶机_取料完成    : BOOL;   // %IX102 (已定义) 打胶机已完成边框抓取
    i_b打胶机_故障        : BOOL;   // %IX77  占位符: 打胶机设备故障报警
    i_b打胶机_急停        : BOOL;   // %IX78  占位符: 打胶机急停状态
    i_b打胶机_通讯异常    : BOOL;   // %IX79  占位符: 与打胶机通讯中断

    (*--- 打胶机输出信号 (到CPU本体DO, 硬接线/通讯) ---*)
    q_b打胶机_请求运行    : BOOL;   // -> Y40 占位符: 请求打胶机启动运行
    q_b允许抓料            : BOOL;   // -> Y44  (已定义) 通知打胶机可以抓取边框
    q_b安全区信号          : BOOL;   // -> Y47  (已定义) 安全区开放/关闭信号
    q_b打胶机_复位请求    : BOOL;   // -> Y41 占位符: 向打胶机发送复位请求

    // ==========================================================================
    // 六点五、组框机信号映射 (上游设备: 提供边框)
    // ==========================================================================

    (*--- 组框机输入信号 (来自CPU本体DI, 地址预留) ---*)
    i_b组框机_自动中      : BOOL;   // 占位符: 组框机自动运行中
    i_b组框机_允许送料    : BOOL;   // 占位符: 组框机允许向缓存机输送边框
    i_b组框机_有料请求    : BOOL;   // 占位符: 组框机有边框需要送入缓存机
    i_b组框机_开门请求    : BOOL;   // 占位符: 组框机操作门打开(需本机暂停)
    i_b组框机_急停        : BOOL;   // 占位符: 组框机急停信号(需联锁)
    i_b组框机_安全异常    : BOOL;   // 占位符: 组框机安全系统异常
    i_b组框机_通讯异常    : BOOL;   // 占位符: 与组框机通讯异常

    (*--- 组框机输出信号 (到CPU本体DO, 地址预留) ---*)
    q_b组框机_请求送料    : BOOL;   // 占位符: 向组框机请求输送边框
    q_b组框机_暂停          : BOOL;   // 占位符: 向组框机发送暂停指令
    q_b组框机_急停          : BOOL;   // 占位符: 向组框机发送急停联锁信号
    q_b申请开门             : BOOL;   // 占位符: 向组框机申请开门操作
    q_b组框机_就绪          : BOOL;   // 占位符: 本机就绪, 可接收边框

    // ==========================================================================
    // 七、HMI数据 - 输入 (M/D区读取 -> 逻辑变量)
    // 注: 具体M/D地址需根据HMI画面分配表确定, 此处使用占位符
    // ==========================================================================

    (*--- 模式选择 (互斥信号) ---*)
    bHMI_自动模式       : BOOL;   // M?  (自动运行模式选择)
    bHMI_手动模式       : BOOL;   // M?  (手动调试模式选择)

    (*--- 操作按钮 ---*)
    bHMI_启动           : BOOL;   // M?  (启动按钮, 上升沿触发)
    bHMI_停止           : BOOL;   // M?  (停止按钮, 电平有效)
    bHMI_复位           : BOOL;   // M?  (复位按钮, 电平有效)

    (*--- 工艺参数设定 (REAL类型) ---*)
    rHMI_输送速度设定    : REAL;   // D?  (输送带速度设定 Hz或m/min)
    rHMI_伺服速度设定    : REAL;   // D?  (伺服轴速度设定 mm/s或%)
    rHMI_取料速度设定    : REAL;   // D?  (取料过程速度 mm/s)
    rHMI_放料速度设定    : REAL;   // D?  (放料过程速度 mm/s)

    (*--- 动作时间参数设定 (INT类型, 单位ms) ---*)
    iHMI_分料时间设定    : INT;    // D?  (分料动作保持时间)
    iHMI_夹紧确认时间设定 : INT;   // D?  (夹爪夹紧确认等待时间)
    iHMI_升降动作时间设定 : INT;   // D?  (升降气缸动作超时时间)

    // ==========================================================================
    // 八、HMI数据 - 输出 (逻辑变量 -> M/D区回写)
    // ==========================================================================

    (*--- 系统状态显示 ---*)
    bHMI_系统运行中      : BOOL;   // -> M?  (系统正在自动运行)
    bHMI_系统故障        : BOOL;   // -> M?  (系统有故障)
    bHMI_系统就绪        : BOOL;   // -> M?  (系统初始化完成, 可启动)

    (*--- 各工站运行状态 ---*)
    bHMI_输送机运行中    : BOOL;   // -> M?  (四层输送机运行中)
    bHMI_取放料运行中    : BOOL;   // -> M?  (取放料机构运行中)
    bHMI_送料机构运行中  : BOOL;   // -> M?  (打胶机送料机构运行中)

    (*--- 报警信息显示 ---*)
    iHMI_全局报警代码    : INT;    // -> D?  (当前最高优先级报警码)
    wHMI_全局报警字      : WORD;   // -> D?  (全局报警字, 位或组合)
    bHMI_任何报警激活    : BOOL;   // -> M?  (是否有任何报警激活)

    (*--- 取放料位置显示 ---*)
    iHMI_当前取料层数    : INT;    // -> D?  (当前正在处理的层数 0~4)
    iHMI_取放料步序      : INT;    // -> D?  (取放料状态机步序 0~10)

    // ==========================================================================
    // 九、中间变量 (用于工站间信号传递和内部计算)
    // ==========================================================================

    (*--- 下游信号传递 (工站间的协调信号) ---*)
    (* 四层输送机 -> 取放料机构: 放料完成通知 *)
    b输送机_L1_放料完成  : BOOL;   // 第1层放料完成, 可取料
    b输送机_L2_放料完成  : BOOL;   // 第2层放料完成, 可取料
    b输送机_L3_放料完成  : BOOL;   // 第3层放料完成, 可取料
    b输送机_L4_放料完成  : BOOL;   // 第4层放料完成, 可取料

    (* 取放料机构 -> 打胶机送料机构: 放料完成通知 *)
    b取放料_放料完成    : BOOL;   // 取放料机构完成放料, 送料机构可工作

    (*--- 系统使能标志 (用于统一控制各工站的使能信号) ---*)
    b系统使能            : BOOL;   // 系统总使能(安全条件满足后置TRUE)

    (*--- 外部设备联锁标志 ---*)
    b组框机紧急停止      : BOOL;   // 组框机急停/安全异常时强制本机停止
    i_外部设备报警汇总   : INT;    // 外部设备故障报警码(300~399段, 供公共报警FB)

    (*--- 手动操作信号缓存 (14个手动操作BOOL, 来自HMI) ---*)
    (* 四层输送机手动操作 (24个: 4层×6操作) ---*)
    i_bLx_阻挡下降         : ARRAY[1..4] OF BOOL;
    i_bLx_阻挡上升         : ARRAY[1..4] OF BOOL;
    i_bLx_分料推出         : ARRAY[1..4] OF BOOL;
    i_bLx_分料复位         : ARRAY[1..4] OF BOOL;
    i_bLx_输送正转         : ARRAY[1..4] OF BOOL;
    i_bLx_输送反转         : ARRAY[1..4] OF BOOL;

    (* 取放料机构手动操作 (14个) ---*)
    b_Z轴点动上          : BOOL;
    b_Z轴点动下          : BOOL;
    b_X1轴点动前         : BOOL;
    b_X1轴点动后         : BOOL;
    b_升降上升           : BOOL;
    b_升降下降           : BOOL;
    b_前夹紧夹紧         : BOOL;
    b_前夹紧松开         : BOOL;
    b_后夹紧夹紧         : BOOL;
    b_后夹紧松开         : BOOL;
    b_前夹紧2夹紧        : BOOL;
    b_前夹紧2松开        : BOOL;
    b_后夹紧2夹紧        : BOOL;
    b_后夹紧2松开        : BOOL;

    (* 打胶机送料机构手动操作 (2个) ---*)
    b_X2轴点动前         : BOOL;
    b_X2轴点动后         : BOOL;

    (*--- 安全系统输入 (来自CPU本体DI) ---*)
    i_b急停按钮            : BOOL;   // X16 (操作台急停按钮)
    b复位按钮            : BOOL;   // X17 (操作台复位按钮)
    i_b前门锁定            : BOOL;   // X15 (前安全门锁定状态)
    i_b后门锁定            : BOOL;   // X14 (后安全门锁定状态)

    (*--- 安全系统输出 (到CPU本体DO) ---*)
    q_b安全继电器启动      : BOOL;   // -> Y13 (安全继电器启动信号)

    (*--- 工站报警代码变量 ---*)
    i_ConveyorAlarm       : INT;    // 四层输送机报警代码
    i_PickPlaceAlarm      : INT;    // 取放料机构报警代码
    i_GlueMachineAlarm    : INT;    // 打胶机送料机构报警代码

    (*--- MES相关变量 ---*)
    iMES报警计数         : INT;    // 自上次复位以来的累计报警次数
    iMES报警队列         : ARRAY[0..9] OF INT;  // 最近10条报警记录(去重后)
    b新报警检测到        : BOOL;   // 新报警脉冲标志(触发MES上传)
END_VAR

//==============================================================================
// 主程序执行体 (严格按照10步顺序执行)
//==============================================================================

//==============================================================================
// Step1: IO映射输入 (X地址 -> 逻辑变量)
// 说明: 将所有物理输入地址映射到逻辑变量, 供后续功能块使用
//       此步骤确保功能块完全不依赖物理地址, 实现硬件解耦
//==============================================================================

// 1.1 CPU本体输入映射 (伺服/安全/打胶机信号)
i_bZ轴_原点           := %IX0;       // Z轴原点传感器
i_bX1轴_原点          := %IX1;       // X1轴原点传感器
i_bX2轴_原点          := %IX2;       // X2轴原点传感器
i_bZ轴_正向限位       := %IX3;       // Z轴正向限位
i_bZ轴_反向限位       := %IX4;       // Z轴反向限位
i_bX1轴_正向限位      := %IX5;       // X1轴正向限位
i_bX1轴_反向限位      := %IX6;       // X1轴反向限位
i_bX2轴_正向限位      := %IX7;       // X2轴正向限位
i_bX2轴_反向限位      := %IX10;      // X2轴反向限位
i_bZ轴_伺服故障       := %IX11;      // Z轴伺服故障报警
i_bX1轴_伺服故障      := %IX12;      // X1轴伺服故障报警
i_bX2轴_伺服故障      := %IX13;      // X2轴伺服故障报警
i_b前门锁定            := %IX15;      // 前安全门锁定状态
i_b后门锁定            := %IX14;      // 后安全门锁定状态
i_b急停按钮            := %IX16;      // 操作台急停按钮
b复位按钮            := %IX17;      // 操作台复位按钮

// 1.2 打胶机外部信号映射 (下游设备交互)
i_b打胶机_自动中      := %IX75;      // 打胶机自动运行中状态
i_b打胶机_允许送料    := %IX76;      // (已定义) 打胶机允许送料信号
i_b打胶机_取料完成    := %IX102;     // (已定义) 打胶机取料完成信号
i_b打胶机_故障        := FALSE;       // 占位符: 待分配DI地址 (原%IX77可能冲突)
i_b打胶机_急停        := FALSE;       // 占位符: 待分配DI地址
i_b打胶机_通讯异常    := FALSE;       // 占位符: 待分配DI地址(或通讯诊断字)

// 1.2b 组框机外部信号映射 (上游设备交互, 地址预留)
// 注: 组框机信号通过硬接线或总线通讯接入, 具体地址待现场确定
i_b组框机_自动中      := FALSE;       // 占位符: 待分配DI/通讯地址
i_b组框机_允许送料    := FALSE;       // 占位符: 待分配DI/通讯地址
i_b组框机_有料请求    := FALSE;       // 占位符: 待分配DI/通讯地址
i_b组框机_开门请求    := FALSE;       // 占位符: 待分配DI/通讯地址
i_b组框机_急停        := FALSE;       // 占位符: 待分配DI/通讯地址(安全联锁)
i_b组框机_安全异常    := FALSE;       // 占位符: 待分配DI/通讯地址
i_b组框机_通讯异常    := FALSE;       // 占位符: 待分配DI/通讯地址(或通讯诊断)

// 1.3 DI扩展模块3映射 (4层L4 + 3层L3 分料输入)
// 注: 使用全局软元件地址格式, 具体地址需根据PLC配置确认
// DI3:X0 = 4层分料前感应器 (索引[4])
i_bLx_分料前感应器[4] := %IX51;      // DI3:X0 -> L4
i_bLx_到位感应器1[4]  := %IX52;      // DI3:X2 -> L4
i_bLx_到位感应器2[4]  := %IX53;      // DI3:X3 -> L4
i_bLx_阻挡气缸上位[4] := %IX54;      // DI3:X4 -> L4
i_bLx_阻挡气缸下位[4] := %IX55;      // DI3:X5 -> L4
i_bLx_分料气缸上位[4] := %IX56;      // DI3:X6 -> L4
i_bLx_分料气缸下位[4] := %IX57;      // DI3:X7 -> L4

// DI3:X10-X17 = 3层L3 分料输入
i_bLx_分料前感应器[3] := %IX61;      // DI3:X11 -> L3
i_bLx_到位感应器1[3]  := %IX62;      // DI3:X12 -> L3
i_bLx_到位感应器2[3]  := %IX63;      // DI3:X13 -> L3
i_bLx_阻挡气缸上位[3] := %IX64;      // DI3:X14 -> L3
i_bLx_阻挡气缸下位[3] := %IX65;      // DI3:X15 -> L3
i_bLx_分料气缸上位[3] := %IX66;      // DI3:X16 -> L3
i_bLx_分料气缸下位[3] := %IX67;      // DI3:X17 -> L3

// 1.4 DI扩展模块4映射 (2层L2 + 1层L1 分料输入)
// DI4:X0-X7 = 2层L2 分料输入
i_bLx_分料前感应器[2] := %IX71;      // DI4:X1 -> L2
i_bLx_到位感应器1[2]  := %IX72;      // DI4:X2 -> L2
i_bLx_到位感应器2[2]  := %IX73;      // DI4:X3 -> L2
i_bLx_阻挡气缸上位[2] := %IX74;      // DI4:X4 -> L2
i_bLx_阻挡气缸下位[2] := %IX75;      // DI4:X5 -> L2
i_bLx_分料气缸上位[2] := %IX76;      // DI4:X6 -> L2
i_bLx_分料气缸下位[2] := %IX77;      // DI4:X7 -> L2

// DI4:X10-X17 = 1层L1 分料输入
i_bLx_分料前感应器[1] := %IX81;      // DI4:X11 -> L1
i_bLx_到位感应器1[1]  := %IX82;      // DI4:X12 -> L1
i_bLx_到位感应器2[1]  := %IX83;      // DI4:X13 -> L1
i_bLx_阻挡气缸上位[1] := %IX84;      // DI4:X14 -> L1
i_bLx_阻挡气缸下位[1] := %IX85;      // DI4:X15 -> L1
i_bLx_分料气缸上位[1] := %IX86;      // DI4:X16 -> L1
i_bLx_分料气缸下位[1] := %IX87;      // DI4:X17 -> L1

// 1.5 远程IO_1输入映射 (取放料机构气缸传感器 + 产品检测)
// 注: CC-Link Basic站号1, 地址为相对于该站的偏移量
i_b升降_动点          := %IX100;     // Remote_X0 (升降气缸动点)
i_b升降_原点          := %IX101;     // Remote_X1 (升降气缸原点)
i_b前夹紧_动点        := %IX102;     // Remote_X2 (前夹紧动点)
i_b前夹紧_原点        := %IX103;     // Remote_X3 (前夹紧原点)
i_b后夹紧_动点        := %IX104;     // Remote_X4 (后夹紧动点)
i_b后夹紧_原点        := %IX105;     // Remote_X5 (后夹紧原点)
i_b前夹紧2_动点       := %IX106;     // Remote_X6 (前夹紧2动点)
i_b前夹紧2_原点       := %IX107;     // Remote_X7 (前夹紧2原点)
i_b后夹紧2_动点       := %IX108;     // Remote_X8 (后夹紧2动点)
i_b后夹紧2_原点       := %IX109;     // Remote_X9 (后夹紧2原点)
i_b长边1检测          := %IX110;     // Remote_XC (长边1光电)
i_b长边2检测          := %IX111;     // Remote_XD (长边2光电)
i_b短边1检测          := %IX112;     // Remote_XE (短边1光电)
i_b短边2检测          := %IX113;     // Remote_XF (短边2光电)

//==============================================================================
// Step2: HMI数据读取 (M/D区 -> 逻辑变量)
// 说明: 从HMI的操作界面读取模式选择、按钮状态、参数设定值
//       这些数据将作为各工站的输入参数传入
//==============================================================================

// 2.1 模式选择信号 (互斥, 来自HMI M区)
bHMI_自动模式       := %MX0;       // 占位符: 自动模式选择
bHMI_手动模式       := %MX1;       // 占位符: 手动模式选择

// 2.2 操作按钮 (来自HMI M区)
bHMI_启动           := %MX2;       // 占位符: 启动按钮
bHMI_停止           := %MX3;       // 占位符: 停止按钮
bHMI_复位           := %MX4;       // 占位符: 复位按钮

// 2.3 工艺参数设定 (REAL类型, 来自HMI D区)
rHMI_输送速度设定    := %DW100;     // 占位符: 输送带速度设定
rHMI_伺服速度设定    := %DW102;     // 占位符: 伺服轴速度设定
rHMI_取料速度设定    := %DW104;     // 占位符: 取料过程速度
rHMI_放料速度设定    := %DW106;     // 占位符: 放料过程速度

// 2.4 动作时间参数设定 (INT类型, 来自HMI D区)
iHMI_分料时间设定    := %DW108;     // 占位符: 分料动作保持时间(ms)
iHMI_夹紧确认时间设定 := %DW110;    // 占位符: 夹紧确认时间(ms)
iHMI_升降动作时间设定 := %DW112;    // 占位符: 升降动作超时时间(ms)

// 2.5 手动操作信号 (从HMI M区读取, 用于手动模式下对各机构的点动控制)
// 注: 具体M地址需根据HMI画面设计确定, 此处使用占位符
(* 四层输送机手动操作: 每层6个操作, 共24个BOOL *)
i_bLx_阻挡下降[1]     := %MX10;      // L1阻挡下降
i_bLx_阻挡上升[1]     := %MX11;      // L1阻挡上升
i_bLx_分料推出[1]     := %MX12;      // L1分料推出
i_bLx_分料复位[1]     := %MX13;      // L1分料复位
i_bLx_输送正转[1]     := %MX14;      // L1输送正转
i_bLx_输送反转[1]     := %MX15;      // L1输送反转

i_bLx_阻挡下降[2]     := %MX16;      // L2阻挡下降
i_bLx_阻挡上升[2]     := %MX17;      // L2阻挡上升
i_bLx_分料推出[2]     := %MX18;      // L2分料推出
i_bLx_分料复位[2]     := %MX19;      // L2分料复位
i_bLx_输送正转[2]     := %MX20;      // L2输送正转
i_bLx_输送反转[2]     := %MX21;      // L2输送反转

i_bLx_阻挡下降[3]     := %MX22;      // L3阻挡下降
i_bLx_阻挡上升[3]     := %MX23;      // L3阻挡上升
i_bLx_分料推出[3]     := %MX24;      // L3分料推出
i_bLx_分料复位[3]     := %MX25;      // L3分料复位
i_bLx_输送正转[3]     := %MX26;      // L3输送正转
i_bLx_输送反转[3]     := %MX27;      // L3输送反转

i_bLx_阻挡下降[4]     := %MX28;      // L4阻挡下降
i_bLx_阻挡上升[4]     := %MX29;      // L4阻挡上升
i_bLx_分料推出[4]     := %MX30;      // L4分料推出
i_bLx_分料复位[4]     := %MX31;      // L4分料复位
i_bLx_输送正转[4]     := %MX32;      // L4输送正转
i_bLx_输送反转[4]     := %MX33;      // L4输送反转

(* 取放料机构手动操作: 14个BOOL *)
b_Z轴点动上          := %MX34;      // Z轴向上点动
b_Z轴点动下          := %MX35;      // Z轴向下点动
b_X1轴点动前         := %MX36;      // X1轴向前点动
b_X1轴点动后         := %MX37;      // X1轴向后点动
b_升降上升           := %MX38;      // 升降气缸上升
b_升降下降           := %MX39;      // 升降气缸下降
b_前夹紧夹紧         := %MX40;      // 前夹紧夹紧
b_前夹紧松开         := %MX41;      // 前夹紧松开
b_后夹紧夹紧         := %MX42;      // 后夹紧夹紧
b_后夹紧松开         := %MX43;      // 后夹紧松开
b_前夹紧2夹紧        := %MX44;      // 前夹紧2夹紧
b_前夹紧2松开        := %MX45;      // 前夹紧2松开
b_后夹紧2夹紧        := %MX46;      // 后夹紧2夹紧
b_后夹紧2松开        := %MX47;      // 后夹紧2松开

(* 打胶机送料机构手动操作: 2个BOOL *)
b_X2轴点动前         := %MX48;      // X2轴向前点动
b_X2轴点动后         := %MX49;      // X2轴向后点动

//==============================================================================
// Step3: 外部设备信号处理 (打胶机/组框机交互信号预处理)
// 说明:
//   1. 打胶机信号: 有效性检查/通讯诊断/安全回退
//   2. 组框机信号: 安全联锁/开门互锁/请求协调
//   3. 外部设备报警汇总: 统一计算300段报警码供公共报警FB使用
//==============================================================================

// 3.1 打胶机信号有效性检查与安全回退 (S02修复)
// 当通讯异常时, 强制将关键输入信号置为保守值(禁止状态)
IF i_b打胶机_通讯异常 THEN
    i_b打胶机_允许送料 := FALSE;   // 假设不允许送料
    i_b打胶机_取料完成 := FALSE;    // 假设未取料完成
    q_b允许抓料       := FALSE;     // 强制禁止抓料输出
    q_b安全区信号     := FALSE;     // 强制关闭安全区
END_IF;

// 3.2 组框机安全联锁处理 (S04修复: 完整实现)
// 组框机急停/安全异常 -> 本机必须立即停止 + 回传确认
IF i_b组框机_急停 OR i_b组框机_安全异常 THEN
    q_b组框机_急停 := TRUE;          // 向组框机回传急停确认
    b组框机紧急停止 := TRUE;         // 设置本机停止标志(传给各工站)
ELSE
    q_b组框机_急停 := FALSE;
    b组框机紧急停止 := FALSE;
END_IF;

// 组框机开门请求 -> 本机需暂停运行 (互锁)
IF i_b组框机_开门请求 THEN
    q_b组框机_暂停 := TRUE;          // 通知组框机本机已暂停
    q_b申请开门    := TRUE;          // 向组框机确认可以开门
ELSE
    q_b组框机_暂停 := FALSE;
    q_b申请开门    := FALSE;
END_IF;

// 3.3 本机就绪信号生成 (W03修复: 完善条件)
// 就绪 = 自动模式 AND 系统使能 AND 无报警 AND 非紧急停止
q_b组框机_就绪 := bHMI_自动模式
                   AND b系统使能
                   AND (NOT bHMI_任何报警激活)
                   AND (NOT b组框机紧急停止);

// 3.4 送料请求协调逻辑 (W04修复: 取消注释并激活)
// 当本机需要边框且就绪且上游允许时, 请求送料
IF b系统使能
   AND (NOT b组框机紧急停止)         // 无紧急停止
   AND i_b组框机_允许送料             // 上游允许送出
   AND bHMI_自动模式                  // 自动模式下才请求
THEN
    q_b组框机_请求送料 := TRUE;
ELSE
    q_b组框机_请求送料 := FALSE;
END_IF;

// 3.5 打胶机主动控制信号生成 (W01修复: 补充触发逻辑)
// 请求运行: 本机自动启动且打胶机未在自动运行中
IF bHMI_自动模式 AND b系统使能 AND NOT i_b打胶机_自动中 THEN
    q_b打胶机_请求运行 := TRUE;
ELSE
    q_b打胶机_请求运行 := FALSE;
END_IF;

// 复位请求: 本机复位且打胶机有故障或急停
IF (bHMI_复位 OR b复位按钮) AND (i_b打胶机_故障 OR i_b打胶机_急停) THEN
    q_b打胶机_复位请求 := TRUE;
ELSE
    q_b打胶机_复位请求 := FALSE;
END_IF;

// 3.6 外部设备报警码汇总 (W06修复: 新增300段报警)
// 将外部设备故障统一编码, 传入公共报警FB的扩展通道
IF i_b打胶机_故障 THEN
    i_外部设备报警汇总 := 300;        // 300=打胶机设备故障
ELSIF i_b打胶机_急停 THEN
    i_外部设备报警汇总 := 301;        // 301=打胶机急停
ELSIF i_b打胶机_通讯异常 THEN
    i_外部设备报警汇总 := 302;        // 302=打胶机通讯异常
ELSIF i_b组框机_急停 THEN
    i_外部设备报警汇总 := 310;        // 310=组框机急停
ELSIF i_b组框机_安全异常 THEN
    i_外部设备报警汇总 := 311;        // 311=组框机安全系统异常
ELSIF i_b组框机_通讯异常 THEN
    i_外部设备报警汇总 := 312;        // 312=组框机通讯异常
ELSE
    i_外部设备报警汇总 := 0;           // 0=无外部设备报警
END_IF;

//==============================================================================
// Step3.5: 系统使能计算 (W09修复: 提前到工站调用之前)
// 说明: 安全条件满足后置位b系统使能, 供后续Step4~Step6各工站使用
//       包含S01修复: 增加外部设备安全联锁条件
//==============================================================================

(* 安全条件检查(S01修复 - 完整版):
   1. 本机急停按钮未按下 (常闭触点, 正常状态为TRUE)
   2. 前安全门已锁定
   3. 后安全门已锁定
   4. 打胶机无急停且无故障 (新增: 下游设备安全联锁)
   5. 组框机无急停 (新增: 上游设备安全联锁, 预留激活)
*)
IF NOT i_b急停按钮
   AND i_b前门锁定
   AND i_b后门锁定
   AND NOT i_b打胶机_急停              (* S01新增: 打胶机急停联锁 *)
   AND NOT i_b打胶机_故障               (* S01新增: 打胶机故障联锁 *)
   AND NOT i_b组框机_急停               (* S01新增: 组框机急停联锁(预留) *)
THEN
    b系统使能 := TRUE;
    q_b安全继电器启动 := TRUE;
    bHMI_系统就绪 := TRUE;
ELSE
    b系统使能 := FALSE;
    q_b安全继电器启动 := FALSE;
    bHMI_系统就绪 := FALSE;
END_IF;

//==============================================================================
// Step4: 调用fb四层输送机 (工站1: 分料/输送控制)
// 说明: 传入所有传感器输入+HMI控制信号+工艺参数+下游反馈
//       接收所有执行器请求输出+下游信号+状态+报警
// 架构: V4.0.0 容器模式 (内部实例化4个 FB_单层输送机)
// 接口: 外部保持ARRAY[1..4]形式, 内部自动分发到各单层实例
//==============================================================================

fb四层输送机(
    (* 一、系统控制信号 *)
    i_b使能               := b系统使能 AND (NOT b组框机紧急停止),  // S04: 增加组框机联锁
    i_b自动模式           := bHMI_自动模式,
    i_b手动模式           := bHMI_手动模式,
    i_b启动               := bHMI_启动,
    i_b停止               := bHMI_停止,
    i_b复位               := bHMI_复位 OR b复位按钮,

    (* 二、手动操作信号 (每层6个, 共24个) *)
    i_b阻挡下降           := i_bLx_阻挡下降,
    i_b阻挡上升           := i_bLx_阻挡上升,
    i_b分料推出           := i_bLx_分料推出,
    i_b分料复位           := i_bLx_分料复位,
    i_b输送正转           := i_bLx_输送正转,
    i_b输送反转           := i_bLx_输送反转,

    (* 三、工艺参数 *)
    i_r输送速度           := rHMI_输送速度设定,
    i_i分料时间           := iHMI_分料时间设定,
    i_i阻挡等待时间        := iHMI_升降动作时间设定,

    (* 四、传感器输入 (4层×7类=28个) *)
    i_b分料前感应器         := i_bLx_分料前感应器,
    i_b到位感应器1          := i_bLx_到位感应器1,
    i_b到位感应器2          := i_bLx_到位感应器2,
    i_b阻挡气缸上位         := i_bLx_阻挡气缸上位,
    i_b阻挡气缸下位         := i_bLx_阻挡气缸下位,
    i_b分料气缸上位         := i_bLx_分料气缸上位,
    i_b分料气缸下位         := i_bLx_分料气缸下位,

    (* 五、下游反馈信号 (取放料机构已取走该层物料) *)
    i_b取放料完成          :=
    (
        FALSE,  // L1: 暂未连接，后续根据实际取放料完成信号连接
        FALSE,  // L2: 暂未连接，后续根据实际取放料完成信号连接
        FALSE,  // L3: 暂未连接，后续根据实际取放料完成信号连接
        FALSE   // L4: 暂未连接，后续根据实际取放料完成信号连接
    ),

    (* 六、执行器请求输出 (4层×5=20个) -> 映射到物理Y地址 *)
    o_b阻挡电磁阀           => q_bLx_阻挡电磁阀,
    o_b分料电磁阀           => q_bLx_分料电磁阀,
    o_b输送带正转           => q_bLx_输送带正转,
    o_b输送带慢速           => q_bLx_输送带慢速,
    o_b输送带反转           => q_bLx_输送带反转,   // 修正: 输出数组(原错误使用输入数组)

    (* 七、下游信号输出 (给取放料机构) *)
    o_b放料完成            =>
    (
        b输送机_L1_放料完成,
        b输送机_L2_放料完成,
        b输送机_L3_放料完成,
        b输送机_L4_放料完成
    ),

    (* 八、状态/HMI显示输出 *)
    o_b运行中             => bHMI_输送机运行中,
    o_b故障               => ,  (* 可选: 连接到全局故障汇总 *)
    o_i当前状态           => ,  (* 可选: HMI显示用 *)
    o_Lx当前步序           => ,  (* 可选: 每层独立步序显示 *)

    (* 九、报警输出 (给公共报警管理器) *** 必须连接 *** *)
    o_i本站报警代码        => i_ConveyorAlarm
);

//==============================================================================
// Step5: 调用fb取放料机构 (工站2: 取放料控制)
// 说明: 传入含上游信号(四层输送机放料完成)的输入
//       接收执行器请求输出+下游信号(给打胶机送料机构)+状态+报警
//==============================================================================

fb取放料机构(
    (* 一、系统控制信号 *)
    i_b使能               := b系统使能 AND (NOT b组框机紧急停止),  // S04: 增加组框机联锁
    i_b自动模式           := bHMI_自动模式,
    i_b手动模式           := bHMI_手动模式,
    i_b启动               := bHMI_启动,
    i_b停止               := bHMI_停止,
    i_b复位               := bHMI_复位 OR b复位按钮,

    (* 二、手动操作信号 (14个) *)
    i_bZ轴点动上          := b_Z轴点动上,
    i_bZ轴点动下          := b_Z轴点动下,
    i_bX1轴点动前         := b_X1轴点动前,
    i_bX1轴点动后         := b_X1轴点动后,
    i_b升降上升           := b_升降上升,
    i_b升降下降           := b_升降下降,
    i_b前夹紧夹紧         := b_前夹紧夹紧,
    i_b前夹紧松开         := b_前夹紧松开,
    i_b后夹紧夹紧         := b_后夹紧夹紧,
    i_b后夹紧松开         := b_后夹紧松开,
    i_b前夹紧2夹紧        := b_前夹紧2夹紧,
    i_b前夹紧2松开        := b_前夹紧2松开,
    i_b后夹紧2夹紧        := b_后夹紧2夹紧,
    i_b后夹紧2松开        := b_后夹紧2松开,

    (* 三、工艺参数 *)
    i_r取料速度           := rHMI_取料速度设定,
    i_r放料速度           := rHMI_放料速度设定,
    i_rZ轴速度            := rHMI_伺服速度设定,
    i_rX1轴速度           := rHMI_伺服速度设定,
    i_i夹紧确认时间       := iHMI_夹紧确认时间设定,
    i_i升降动作时间       := iHMI_升降动作时间设定,

    (* 四、传感器输入 (26个) *)
    (* 气缸位置传感器 (10个) *)
    i_升降_动点           := i_b升降_动点,
    i_升降_原点           := i_b升降_原点,
    i_前夹紧_动点         := i_b前夹紧_动点,
    i_前夹紧_原点         := i_b前夹紧_原点,
    i_后夹紧_动点         := i_b后夹紧_动点,
    i_后夹紧_原点         := i_b后夹紧_原点,
    i_前夹紧2_动点        := i_b前夹紧2_动点,
    i_前夹紧2_原点        := i_b前夹紧2_原点,
    i_后夹紧2_动点        := i_b后夹紧2_动点,
    i_后夹紧2_原点        := i_b后夹紧2_原点,

    (* 产品检测传感器 (4个) *)
    i_长边1检测           := i_b长边1检测,
    i_长边2检测           := i_b长边2检测,
    i_短边1检测           := i_b短边1检测,
    i_短边2检测           := i_b短边2检测,

    (* 伺服轴状态信号 (12个) *)
    i_Z轴_原点            := i_bZ轴_原点,
    i_X1轴_原点           := i_bX1轴_原点,
    i_X2轴_原点           := i_bX2轴_原点,
    i_Z轴_伺服故障        := i_bZ轴_伺服故障,
    i_X1轴_伺服故障       := i_bX1轴_伺服故障,
    i_X2轴_伺服故障       := i_bX2轴_伺服故障,
    i_Z轴_正向限位        := i_bZ轴_正向限位,
    i_Z轴_反向限位        := i_bZ轴_反向限位,
    i_X1轴_正向限位       := i_bX1轴_正向限位,
    i_X1轴_反向限位       := i_bX1轴_反向限位,
    i_X2轴_正向限位       := i_bX2轴_正向限位,
    i_X2轴_反向限位       := i_bX2轴_反向限位,

    (* 五、上游信号 (来自四层输送机的放料完成信号) *)
    i_输送机_L1_放料完成  := b输送机_L1_放料完成,
    i_输送机_L2_放料完成  := b输送机_L2_放料完成,
    i_输送机_L3_放料完成  := b输送机_L3_放料完成,
    i_输送机_L4_放料完成  := b输送机_L4_放料完成,

    (* 六、执行器请求输出 (给主控映射到Y地址) *)
    (* 六、执行器输出 (给主控IO映射) *)
    o_升降_上升           => q_b升降_上升,
    o_升降_下降           => q_b升降_下降,
    o_前夹紧_夹紧         => q_b前夹紧_夹紧,
    o_前夹紧_松开         => q_b前夹紧_松开,
    o_后夹紧_夹紧         => q_b后夹紧_夹紧,
    o_后夹紧_松开         => q_b后夹紧_松开,

    (* 伺服控制输出 (3个, 仅Z轴) *)
    o_Z轴_脉冲输出        => q_bZ轴_脉冲输出,
    o_Z轴_方向输出        => q_bZ轴_方向输出,
    o_Z轴_伺服使能        => q_bZ轴_伺服使能,

    (* 七、下游信号输出 (给打胶机送料机构) *)
    o_放料完成_给送料机构 => b取放料_放料完成,

    (* 八、状态/HMI显示输出 *)
    o_b运行中             => bHMI_取放料运行中,
    o_b故障               => ,
    o_i当前状态           => iHMI_取放料步序,
    o_rZ轴当前位置        => ,  (* 预留: 需要位置反馈接口 *)
    o_rX1轴当前位置       => ,  (* 预留: 需要位置反馈接口 *)
    o_rX2轴当前位置       => ,  (* 预留: 需要位置反馈接口 *)
    o_i当前取料层数       => iHMI_当前取料层数,

    (* 九、报警输出 (给公共报警管理器) *)
    o_i本站报警代码       => i_PickPlaceAlarm
);

//==============================================================================
// Step6: 调用fb打胶机送料机构 (工站3: 送料控制)
// 说明: 传入含上游信号(取放料机构放料完成)+打胶机交互信号的输入
//       接收执行器请求输出(给打胶机)+状态+报警
//==============================================================================

fb打胶机送料机构(
    (* 一、系统控制信号 *)
    i_b使能               := b系统使能 AND (NOT b组框机紧急停止),  // S04: 增加组框机联锁
    i_b自动模式           := bHMI_自动模式,
    i_b手动模式           := bHMI_手动模式,
    i_b启动               := bHMI_启动,
    i_b停止               := bHMI_停止,
    i_b复位               := bHMI_复位 OR b复位按钮,

    (* 二、手动操作信号 (2个) *)
    i_bX2轴点动前         := b_X2轴点动前,
    i_bX2轴点动后         := b_X2轴点动后,

    (* 三、工艺参数 *)
    i_r送料速度           := rHMI_伺服速度设定,
    i_r待机位置           := 0.0,    (* 占位符: 待机位置坐标 *)
    i_r取料位置           := 0.0,    (* 占位符: 取料位置坐标 *)

    (* 四、传感器输入 (4个, 仅X2轴相关) *)
    i_X2轴_原点           := i_bX2轴_原点,
    i_X2轴_正向限位       := i_bX2轴_正向限位,
    i_X2轴_反向限位       := i_bX2轴_反向限位,
    i_X2轴_伺服故障       := i_bX2轴_伺服故障,

    (* 五、打胶机交互信号 (已由主控做IO映射和预处理) *)
    i_打胶机允许送料      := i_b打胶机_允许送料,
    i_打胶机取料完成      := i_b打胶机_取料完成,
    (* 扩展信号 (预留接口, 当前版本可能未使用) *)
    (* i_打胶机自动中     := i_b打胶机_自动中,       *)  (* 预留: 打胶机运行状态互锁 *)
    (* i_打胶机故障       := i_b打胶机_故障,         *)  (* 预留: 打胶机故障联锁 *)

    (* 六、上游信号 (来自取放料机构的放料完成信号) *)
    i_取放料_放料完成     := b取放料_放料完成,

    (* 七、执行器请求输出 (给主控映射到Y地址) *)
    o_允许抓料            => q_b允许抓料,
    o_安全区信号          => q_b安全区信号,

    (* 八、状态/HMI显示输出 *)
    o_b运行中             => bHMI_送料机构运行中,
    o_b故障               => ,
    o_i当前状态           => ,
    o_rX2轴当前位置       => ,  (* 预留: 需要位置反馈接口 *)

    (* 九、报警输出 (给公共报警管理器) *)
    o_i本站报警代码       => i_GlueMachineAlarm
);

//==============================================================================
// Step7: 调用fb公共报警 (工站4: 报警汇总管理)
// 说明: 汇聚三工站的报警代码, 计算全局报警字和最高优先级报警码
//       维护MES报警队列(最近10条去重记录), 产生新报警脉冲标志
//==============================================================================

fb公共报警(
    (* 一、工站报警代码输入 (来自各工站的o_i本站报警代码) *)
    i_i输送机报警        := i_ConveyorAlarm,  (* 来自fb四层输送机.o_i本站报警代码 *)
    i_i取放料报警        := i_PickPlaceAlarm,  (* 来自fb取放料机构.o_i本站报警代码 *)
    i_i送料机构报警      := i_GlueMachineAlarm,  (* 来自fb打胶机送料机构.o_i本站报警代码 *)

    (* 二、操作控制输入 *)
    i_b复位              := bHMI_复位 OR b复位按钮,

    (* 三、HMI显示输出 (由主控写入D区) *)
    o_w全局报警字        => wHMI_全局报警字,
    o_i当前报警代码       => iHMI_全局报警代码,
    o_b任何报警激活       => bHMI_任何报警激活,

    (* 四、MES数据接口输出 *)
    o_iMES报警计数        => iMES报警计数,
    o_iMES报警队列         => iMES报警队列,
    o_b新报警标志          => b新报警检测到
);

(* 将公共报警的全局故障信号同步到HMI故障显示 *)
bHMI_系统故障 := bHMI_任何报警激活;

//==============================================================================
// Step8: IO映射输出 (逻辑变量 -> Y地址)
// 说明: 将各工站的执行器请求输出映射到物理输出地址
//       此步骤确保功能块的逻辑输出能够驱动实际硬件
//==============================================================================

// 8.1 CPU本体输出映射 (伺服脉冲/方向/励磁 + 安全 + 打胶机/组框机信号)
%QY0                := q_bZ轴_脉冲输出;      // Y0: Z轴脉冲输出(PULSE+)
%QY4                := q_bZ轴_方向输出;      // Y4: Z轴方向控制(SIGN+)
%QY10               := q_bZ轴_伺服使能;       // Y10: Z轴伺服励磁(SON)
%QY13               := q_b安全继电器启动;     // Y13: 安全继电器启动

// 8.1b 打胶机输出信号映射 (下游设备交互)
// 注: Y50/Y51避开DO2模块范围(Y32-Y43=DO2), 防止与L1输送带冲突
%QY50               := q_b打胶机_请求运行;    // 占位符: 请求打胶机运行(原Y40冲突,改Y50)
%QY51               := q_b打胶机_复位请求;    // 占位符: 打胶机复位请求(原Y41冲突,改Y51)
%QY44               := q_b允许抓料;           // (已定义) 允许打胶机抓料
%QY47               := q_b安全区信号;         // (已定义) 打胶机安全区信号

// 8.1c 组框机输出信号映射 (上游设备交互, 地址预留)
// 注: 组框机输出可能通过硬接线或总线通讯, 地址待现场确定
(* %QY?              := q_b组框机_请求送料;    *)  (* 占位符: 待分配DO/通讯地址 *)
(* %QY?              := q_b组框机_暂停;          *)  (* 占位符: 待分配DO/通讯地址 *)
(* %QY?              := q_b组框机_急停;          *)  (* 占位符: 待分配DO/通讯地址 *)
(* %QY?              := q_b申请开门;             *)  (* 占位符: 待分配DO/通讯地址 *)
(* %QY?              := q_b组框机_就绪;          *)  (* 占位符: 待分配DO/通讯地址 *)

// 8.2 DO扩展模块1输出映射 (4层L4 + 3层L3 分料输出)
// DO1: Y0-Y5 = L4, Y10-Y15 = L3
%QY20               := q_bLx_阻挡电磁阀[4];   // DO1:Y0 = L4阻挡电磁阀
%QY21               := q_bLx_分料电磁阀[4];    // DO1:Y1 = L4分料电磁阀
%QY22               := q_bLx_输送带正转[4];    // DO1:Y2 = L4输送带正转
%QY23               := q_bLx_输送带慢速[4];    // DO1:Y3 = L4输送带慢速
// %QY24             := ;                     // DO1:Y4 = L4输送带反转(预留)
// %QY25             := ;                     // DO1:Y5 = L4变频器复位(预留)

%QY26               := q_bLx_阻挡电磁阀[3];   // DO1:Y10 = L3阻挡电磁阀
%QY27               := q_bLx_分料电磁阀[3];    // DO1:Y11 = L3分料电磁阀
%QY28               := q_bLx_输送带正转[3];    // DO1:Y12 = L3输送带正转
%QY29               := q_bLx_输送带慢速[3];    // DO1:Y13 = L3输送带慢速
// %QY30             := ;                     // DO1:Y14 = L3输送带反转(预留)
// %QY31             := ;                     // DO1:Y15 = L3变频器复位(预留)

// 8.3 DO扩展模块2输出映射 (2层L2 + 1层L1 分料输出)
// DO2: Y0-Y5 = L2, Y10-Y15 = L1
%QY32               := q_bLx_阻挡电磁阀[2];   // DO2:Y0 = L2阻挡电磁阀
%QY33               := q_bLx_分料电磁阀[2];    // DO2:Y1 = L2分料电磁阀
%QY34               := q_bLx_输送带正转[2];    // DO2:Y2 = L2输送带正转
%QY35               := q_bLx_输送带慢速[2];    // DO2:Y3 = L2输送带慢速
// %QY36             := ;                     // DO2:Y4 = L2输送带反转(预留)
// %QY37             := ;                     // DO2:Y5 = L2变频器复位(预留)

%QY38               := q_bLx_阻挡电磁阀[1];   // DO2:Y10 = L1阻挡电磁阀
%QY39               := q_bLx_分料电磁阀[1];    // DO2:Y11 = L1分料电磁阀
%QY40               := q_bLx_输送带正转[1];    // DO2:Y12 = L1输送带正转
%QY41               := q_bLx_输送带慢速[1];    // DO2:Y13 = L1输送带慢速
// %QY42             := ;                     // DO2:Y14 = L1输送带反转(预留)
// %QY43             := ;                     // DO2:Y15 = L1变频器复位(预留)

// 8.4 远程IO_1输出映射 (取放料机构电磁阀)
// Remote_IO Y10-Y15 = 取放料机构6个气缸控制
%QY200              := q_b升降_上升;           // Remote_Y10: 升降气缸上升
%QY201              := q_b升降_下降;           // Remote_Y11: 升降气缸下降
%QY202              := q_b前夹紧_夹紧;         // Remote_Y12: 前夹紧气缸夹紧
%QY203              := q_b前夹紧_松开;         // Remote_Y13: 前夹紧气缸松开
%QY204              := q_b后夹紧_夹紧;         // Remote_Y14: 后夹紧气缸夹紧
%QY205              := q_b后夹紧_松开;         // Remote_Y15: 后夹紧气缸松开

//==============================================================================
// Step9: HMI状态回写 (逻辑变量 -> M/D区)
// 说明: 将系统状态、各工站运行状态、报警信息回写到HMI
//       供操作员监控设备运行情况
//==============================================================================

// 9.1 系统状态回写 (M区)
%MX5                := bHMI_系统运行中;      // 系统运行中标志
%MX6                := bHMI_系统故障;        // 系统故障标志
%MX7                := bHMI_系统就绪;        // 系统就绪标志(需根据初始化状态设置)

// 9.2 各工站运行状态回写 (M区) [W07修复: 避开M10/M11手动操作区]
%MX8                := bHMI_输送机运行中;    // 四层输送机运行中
%MX9                := bHMI_取放料运行中;    // 取放料机构运行中
%MX12               := bHMI_送料机构运行中;  // 打胶机送料机构运行中(原M10冲突,改M12)

// 9.3 报警信息回写 (D区)
%MW120              := iHMI_全局报警代码;    // 当前最高优先级报警码
%MW122              := WORD_TO_INT(wHMI_全局报警字);  // 全局报警字(INT形式)
%MX13               := bHMI_任何报警激活;    // 是否有报警激活(原M11冲突,改M13)

// 9.4 取放料位置回写 (D区)
%MW124              := iHMI_当前取料层数;    // 当前取料层数(0~4)
%MW126              := iHMI_取放料步序;      // 取放料状态机步序(0~10)

//==============================================================================
// Step10: 报警D区回写 (公共报警输出 -> D400起始)
// 说明: 将公共报警管理器的详细数据写入固定D区地址
//       供HMI报警画面和MES系统读取
//       D区分配方案:
//         D400: 全局报警字(WORD)
//         D402: 当前最高优先级报警码(INT)
//         D404: MES累计报警次数(INT)
//         D406-D425: MES报警队列(10条×INT, 去重后)
//==============================================================================

// 10.1 全局报警字 -> D400 (WORD类型, HMI报警灯指示用)
%DW400              := wHMI_全局报警字;

// 10.2 当前最高优先级报警码 -> D402 (INT类型, HMI文本显示用)
%DW402              := iHMI_全局报警代码;

// 10.3 MES累计报警次数 -> D404 (INT类型, MES统计用)
%DW404              := iMES报警计数;

// 10.4 MES报警队列 -> D406~D425 (10条INT数组, MES上传用)
%DW406              := iMES报警队列[0];   // 最新一条报警
%DW408              := iMES报警队列[1];
%DW410              := iMES报警队列[2];
%DW412              := iMES报警队列[3];
%DW414              := iMES报警队列[4];
%DW416              := iMES报警队列[5];
%DW418              := iMES报警队列[6];
%DW420              := iMES报警队列[7];
%DW422              := iMES报警队列[8];
%DW424              := iMES报警队列[9];   // 最旧一条报警

//==============================================================================
// [已移除] 系统使能逻辑 (原位置)
// ⚠️ 注意: 此逻辑已移至 Step3.5 (工站调用之前), 确保使用本周期最新值
//       新增了打胶机/组框机的安全联锁条件 (S01修复)
//       保留此注释仅为文档追溯, 实际计算见上方 Step3.5 区域
//==============================================================================

(*
IF NOT i_b急停按钮 AND i_b前门锁定 AND i_b后门锁定 THEN
    b系统使能 := TRUE;
    q_b安全继电器启动 := TRUE;
    bHMI_系统就绪 := TRUE;
ELSE
    b系统使能 := FALSE;
    q_b安全继电器启动 := FALSE;
    bHMI_系统就绪 := FALSE;
END_IF;
*)

//==============================================================================
// 系统运行中状态汇总
// 说明: 综合各工站的运行状态, 判断整个系统是否在自动运行中
//==============================================================================

(* 系统运行中条件: 自动模式 AND 任一工站在运行 AND 系统使能 *)
IF bHMI_自动模式 AND b系统使能 THEN
    IF bHMI_输送机运行中 OR bHMI_取放料运行中 OR bHMI_送料机构运行中 THEN
        bHMI_系统运行中 := TRUE;
    ELSE
        (* 自动模式下但所有工站都空闲, 可能是在等待启动或循环间隙 *)
        bHMI_系统运行中 := FALSE;
    END_IF;
ELSE
    (* 非自动模式或系统未使能, 肯定不在运行中 *)
    bHMI_系统运行中 := FALSE;
END_IF;

//==============================================================================
// 新报警检测处理 (触发MES上传)
// 说明: 当检测到新报警脉冲标志时, 执行MES上传相关操作
//       当前版本仅做标记, 实际上传逻辑可在此处扩展或通过中断实现
//==============================================================================

IF b新报警检测到 THEN
    (* 新报警检测到, 可在此处触发MES上传动作 *)
    (* 例如: 置位MES上传请求标志, 或直接调用MES通信功能块 *)
    (* 当前版本预留, 不实现具体上传逻辑 *)
END_IF;

END_PROGRAM

//==============================================================================
// 程序结束
//==============================================================================
